// Mitsubishi GX Developer project: 12-805_20121015   PLC: FX1N

PROGRAM MAIN
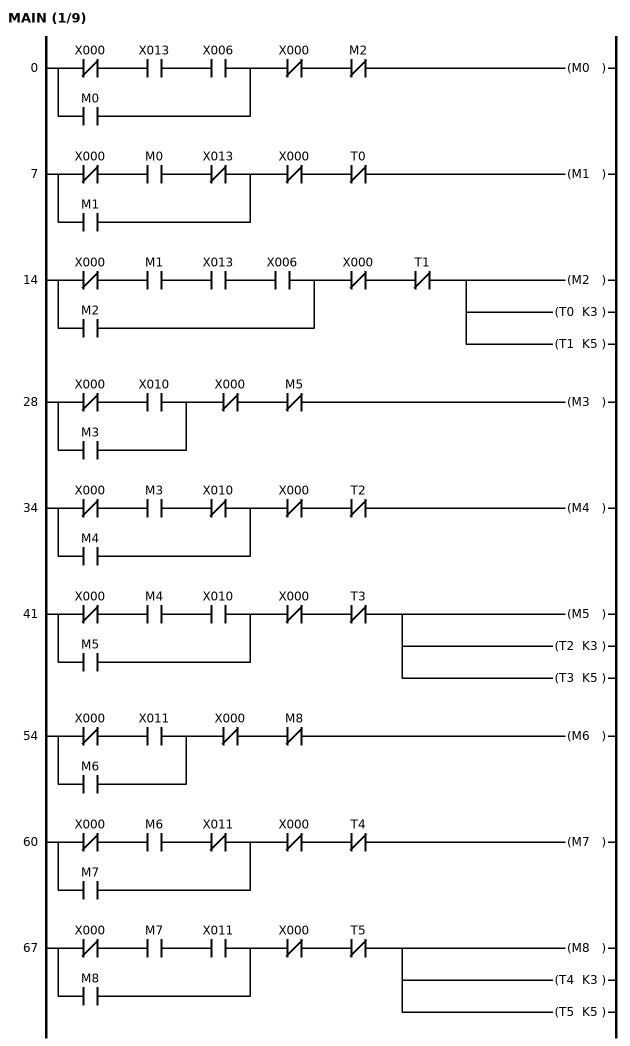
0     LDI     X000
      AND     X013
      AND     X006
      OR      M0
      ANI     X000
      ANI     M2
      OUT     M0
7     LDI     X000
      AND     M0
      ANI     X013
      OR      M1
      ANI     X000
      ANI     T0
      OUT     M1
14    LDI     X000
      AND     M1
      AND     X013
      AND     X006
      OR      M2
      ANI     X000
      ANI     T1
      OUT     M2
      OUT     T0 K3
      OUT     T1 K5
28    LDI     X000
      AND     X010
      OR      M3
      ANI     X000
      ANI     M5
      OUT     M3
34    LDI     X000
      AND     M3
      ANI     X010
      OR      M4
      ANI     X000
      ANI     T2
      OUT     M4
41    LDI     X000
      AND     M4
      AND     X010
      OR      M5
      ANI     X000
      ANI     T3
      OUT     M5
      OUT     T2 K3
      OUT     T3 K5
54    LDI     X000
      AND     X011
      OR      M6
      ANI     X000
      ANI     M8
      OUT     M6
60    LDI     X000
      AND     M6
      ANI     X011
      OR      M7
      ANI     X000
      ANI     T4
      OUT     M7
67    LDI     X000
      AND     M7
      AND     X011
      OR      M8
      ANI     X000
      ANI     T5
      OUT     M8
      OUT     T4 K3
      OUT     T5 K5
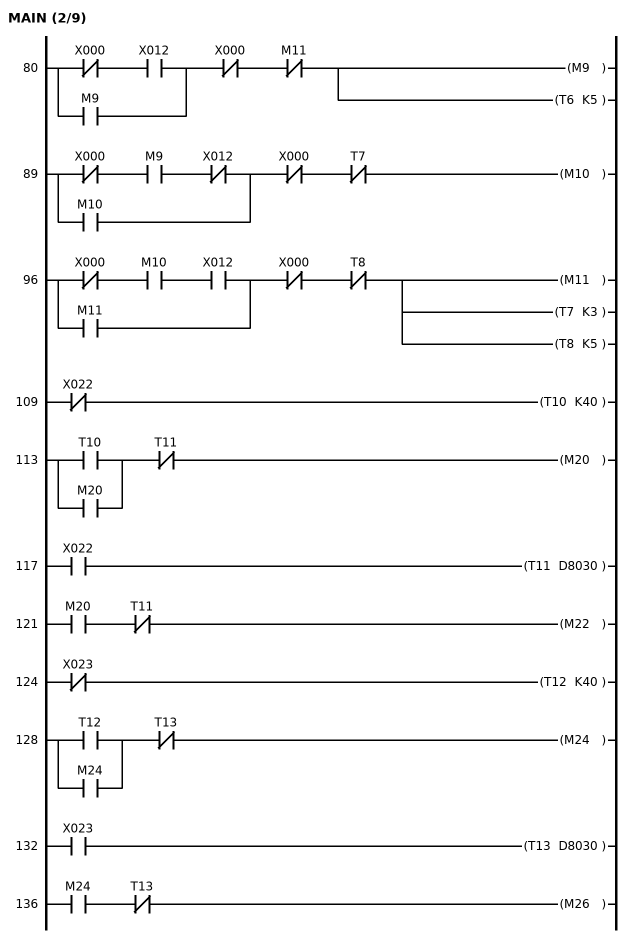
80    LDI     X000
      AND     X012
      OR      M9
      ANI     X000
      ANI     M11
      OUT     M9
      OUT     T6 K5
89    LDI     X000
      AND     M9
      ANI     X012
      OR      M10
      ANI     X000
      ANI     T7
      OUT     M10
96    LDI     X000
      AND     M10
      AND     X012
      OR      M11
      ANI     X000
      ANI     T8
      OUT     M11
      OUT     T7 K3
      OUT     T8 K5
109   LDI     X022
      OUT     T10 K40
113   LD      T10
      OR      M20
      ANI     T11
      OUT     M20
117   LD      X022
      OUT     T11 D8030
121   LD      M20
      ANI     T11
      OUT     M22
124   LDI     X023
      OUT     T12 K40
128   LD      T12
      OR      M24
      ANI     T13
      OUT     M24
132   LD      X023
      OUT     T13 D8030
136   LD      M24
      ANI     T13
      OUT     M26
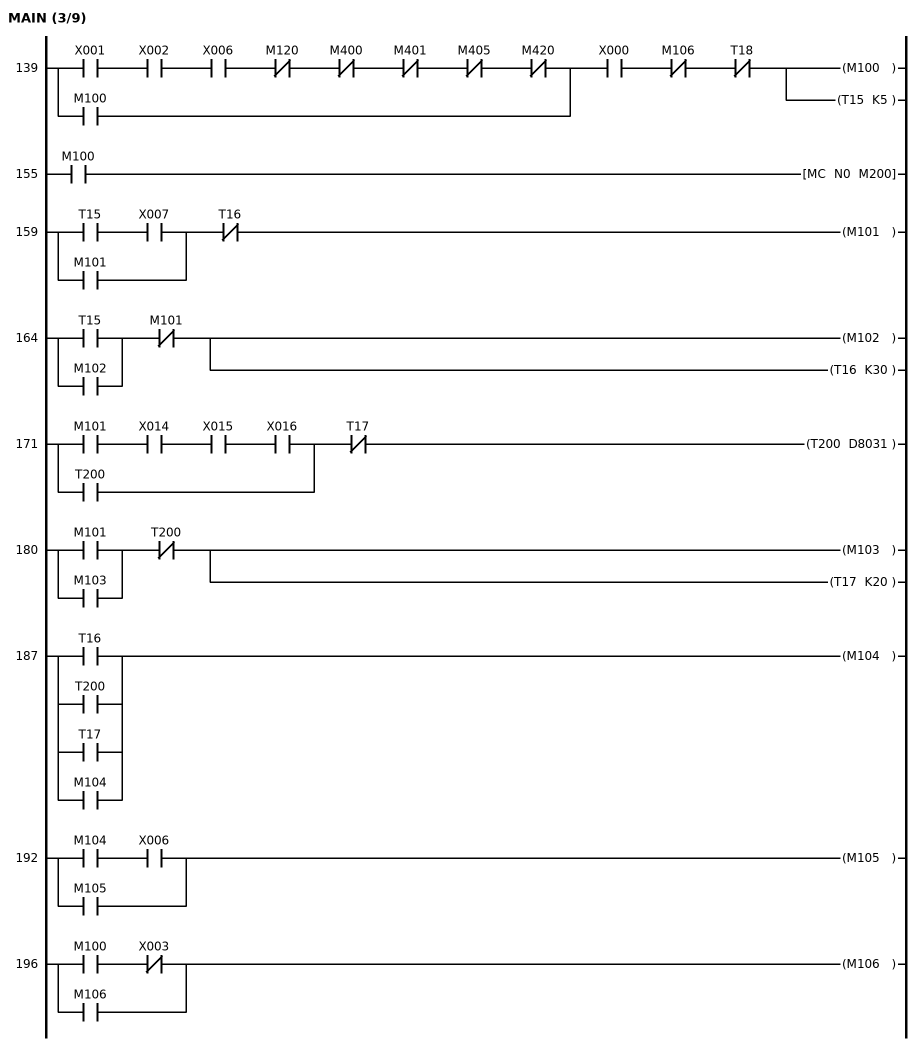
139   LD      X001
      AND     X002
      AND     X006
      ANI     M120
      ANI     M400
      ANI     M401
      ANI     M405
      ANI     M420
      OR      M100
      AND     X000
      ANI     M106
      ANI     T18
      OUT     M100
      OUT     T15 K5
155   LD      M100
      MC      N0 M200
159   LD      T15
      AND     X007
      OR      M101
      ANI     T16
      OUT     M101
164   LD      T15
      OR      M102
      ANI     M101
      OUT     M102
      OUT     T16 K30
171   LD      M101
      AND     X014
      AND     X015
      AND     X016
      OR      T200
      ANI     T17
      OUT     T200 D8031
180   LD      M101
      OR      M103
      ANI     T200
      OUT     M103
      OUT     T17 K20
187   LD      T16
      OR      T200
      OR      T17
      OR      M104
      OUT     M104
192   LD      M104
      AND     X006
      OR      M105
      OUT     M105
196   LD      M100
      ANI     X003
      OR      M106
      OUT     M106
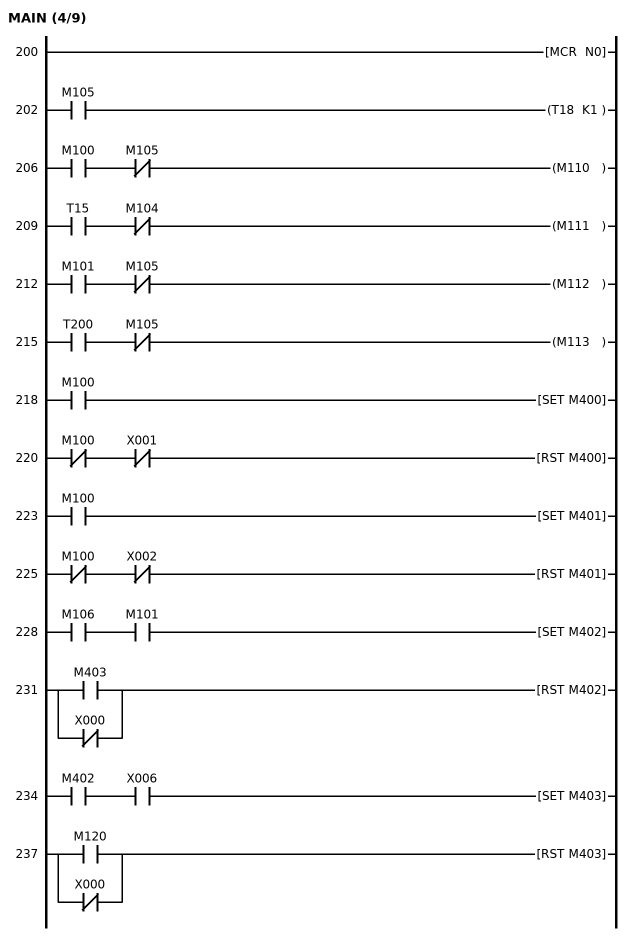
200   MCR     N0
202   LD      M105
      OUT     T18 K1
206   LD      M100
      ANI     M105
      OUT     M110
209   LD      T15
      ANI     M104
      OUT     M111
212   LD      M101
      ANI     M105
      OUT     M112
215   LD      T200
      ANI     M105
      OUT     M113
218   LD      M100
      SET     M400
220   LDI     M100
      ANI     X001
      RST     M400
223   LD      M100
      SET     M401
225   LDI     M100
      ANI     X002
      RST     M401
228   LD      M106
      AND     M101
      SET     M402
231   LD      M403
      ORI     X000
      RST     M402
234   LD      M402
      AND     X006
      SET     M403
237   LD      M120
      ORI     X000
      RST     M403
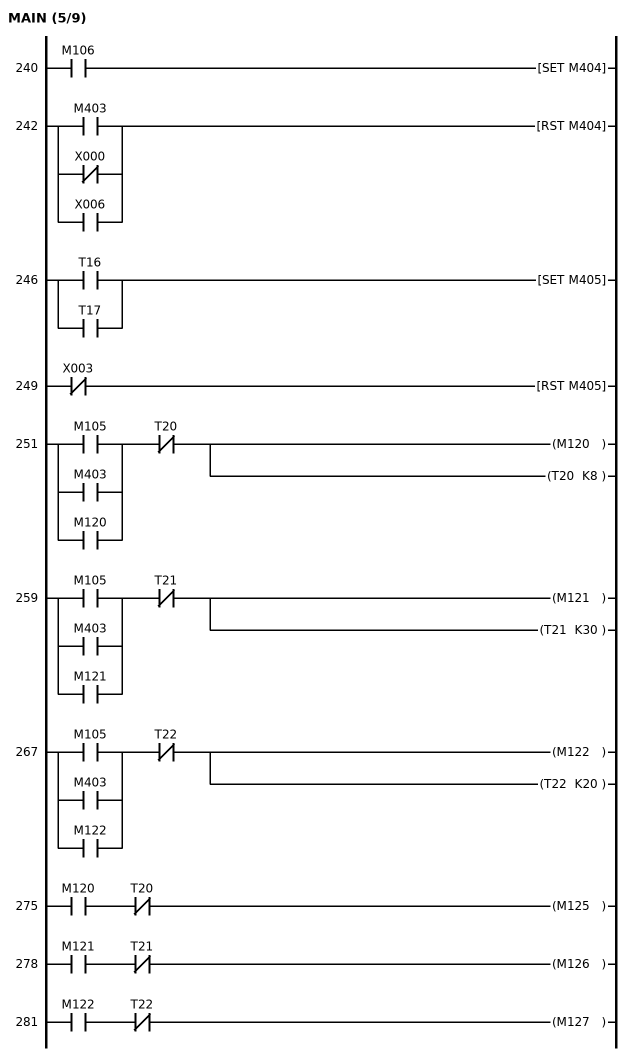
240   LD      M106
      SET     M404
242   LD      M403
      ORI     X000
      OR      X006
      RST     M404
246   LD      T16
      OR      T17
      SET     M405
249   LDI     X003
      RST     M405
251   LD      M105
      OR      M403
      OR      M120
      ANI     T20
      OUT     M120
      OUT     T20 K8
259   LD      M105
      OR      M403
      OR      M121
      ANI     T21
      OUT     M121
      OUT     T21 K30
267   LD      M105
      OR      M403
      OR      M122
      ANI     T22
      OUT     M122
      OUT     T22 K20
275   LD      M120
      ANI     T20
      OUT     M125
278   LD      M121
      ANI     T21
      OUT     M126
281   LD      M122
      ANI     T22
      OUT     M127
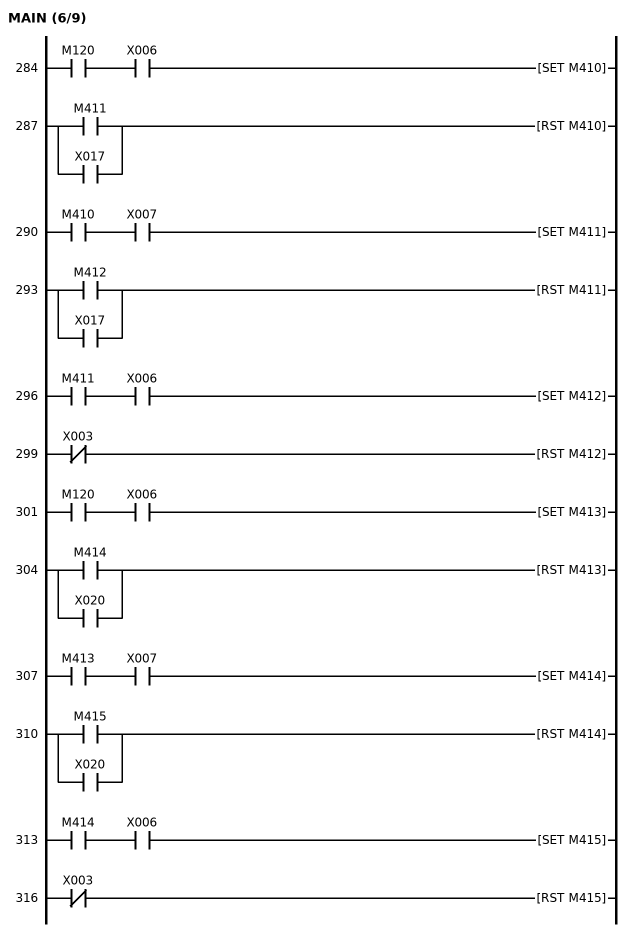
284   LD      M120
      AND     X006
      SET     M410
287   LD      M411
      OR      X017
      RST     M410
290   LD      M410
      AND     X007
      SET     M411
293   LD      M412
      OR      X017
      RST     M411
296   LD      M411
      AND     X006
      SET     M412
299   LDI     X003
      RST     M412
301   LD      M120
      AND     X006
      SET     M413
304   LD      M414
      OR      X020
      RST     M413
307   LD      M413
      AND     X007
      SET     M414
310   LD      M415
      OR      X020
      RST     M414
313   LD      M414
      AND     X006
      SET     M415
316   LDI     X003
      RST     M415
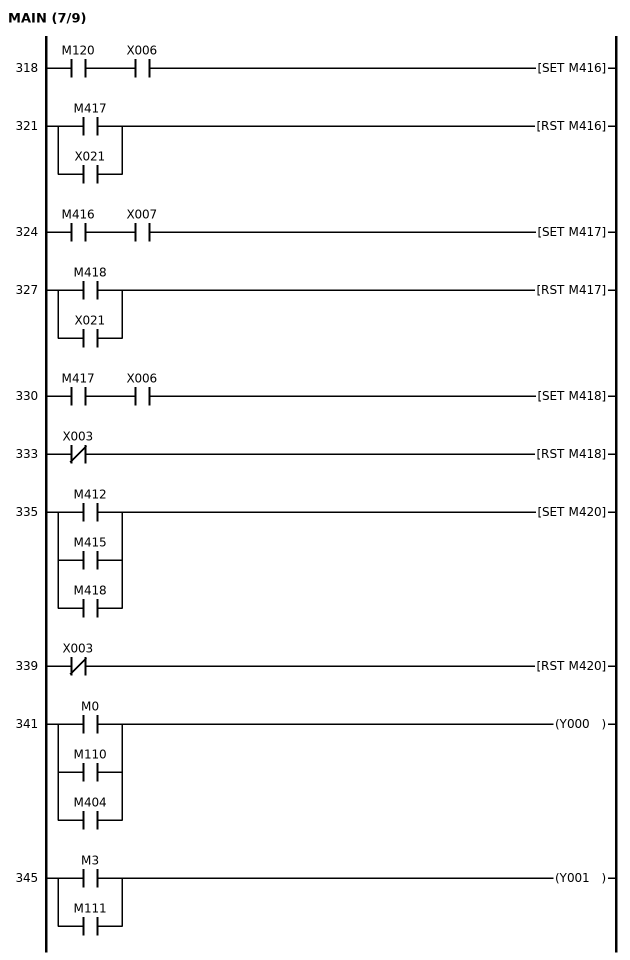
318   LD      M120
      AND     X006
      SET     M416
321   LD      M417
      OR      X021
      RST     M416
324   LD      M416
      AND     X007
      SET     M417
327   LD      M418
      OR      X021
      RST     M417
330   LD      M417
      AND     X006
      SET     M418
333   LDI     X003
      RST     M418
335   LD      M412
      OR      M415
      OR      M418
      SET     M420
339   LDI     X003
      RST     M420
341   LD      M0
      OR      M110
      OR      M404
      OUT     Y000
345   LD      M3
      OR      M111
      OUT     Y001
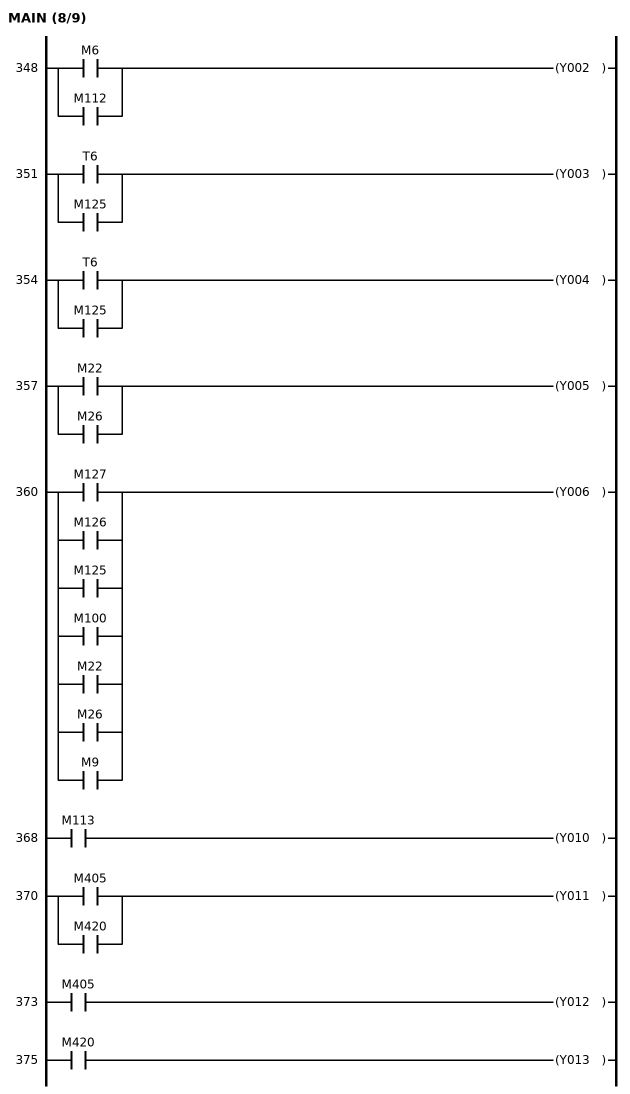
348   LD      M6
      OR      M112
      OUT     Y002
351   LD      T6
      OR      M125
      OUT     Y003
354   LD      T6
      OR      M125
      OUT     Y004
357   LD      M22
      OR      M26
      OUT     Y005
360   LD      M127
      OR      M126
      OR      M125
      OR      M100
      OR      M22
      OR      M26
      OR      M9
      OUT     Y006
368   LD      M113
      OUT     Y010
370   LD      M405
      OR      M420
      OUT     Y011
373   LD      M405
      OUT     Y012
375   LD      M420
      OUT     Y013
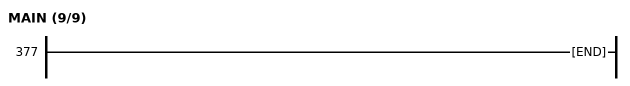
377   END
END_PROGRAM
